FUNCTION_BLOCK FB_AutoStrategy IMPLEMENTS I_ModeStrategy
VAR
	 tonSettle : TON;
      bActive   : BOOL := FALSE;
END_VAR

tonSettle(IN := bActive, PT := GVL_Constants.SETTLE_DELAY);

METHOD GetModeName : STRING
  GetModeName := 'AUTO';
END_METHOD

METHOD Reset
bActive := FALSE;
tonSettle(IN := FALSE, PT := GVL_Constants.SETTLE_DELAY);
END_METHOD

METHOD ShouldLoop : BOOL
ShouldLoop := TRUE;
END_METHOD

END_FUNCTION_BLOCK

(* stored: Version 1.1.0.1, ProductVersion 3.1.4024.16
   POU FB_AutoStrategy: Id {92958d9f-2868-466d-8332-831fb6527921}, SpecialFunc None
   Method GetModeName: Id {a0141eda-8943-49d6-8ed4-d5430a879611}
   Method Reset: Id {6b96ff0a-cddf-435d-b637-3a5c3cd5883c}
   Method ShouldLoop: Id {4cd0e494-3331-4504-922d-c261c3f5c61c} *)
